{attribute 'GeneratedUsingTerminal: EJ7041-0052-0016'}
{attribute addProperty BoxType "EJ7041-0052-0016"}
{attribute addProperty Id "ENC_Status_compactAT %I*ENC_Status_compact_3C6E2C4411STM_StatusAT %I*STM_Status_36ED096F11ENC_Control_compactAT %Q*ENC_Control_compact_2E82BC435STM_ControlAT %Q*STM_Control_5A8B50163STM_VelocityAT %Q*STM_Velocity_A47A3F412WcStateAT %I*WcState_9091E0EB2InfoDataAT %I*InfoData_6538CF5F12"}
{attribute addProperty CRC "36390916"}
{attribute addProperty Size "46"}
TYPE EJ7041_022B4804 EXTENDS EtcSlaveTerminalBase_947E5A46 :
STRUCT
	{attribute addProperty Name "ENC_Status_compact"}
	ENC_Status_compact : ENC_Status_compact_3C6E2C44;
	{attribute addProperty Name "STM_Status"}
	STM_Status : STM_Status_36ED096F;
	{attribute addProperty Name "ENC_Control_compact"}
	ENC_Control_compact : ENC_Control_compact_2E82BC43;
	{attribute addProperty Name "STM_Control"}
	STM_Control : STM_Control_5A8B5016;
	{attribute addProperty Name "STM_Velocity"}
	STM_Velocity : STM_Velocity_A47A3F41;
	{attribute addProperty Name "WcState"}
	WcState : WcState_9091E0EB;
	{attribute addProperty Name "InfoData"}
	InfoData : InfoData_6538CF5F;
END_STRUCT
END_TYPE

(* stored: Version 1.2.0.0, ProductVersion 3.1.4024.9
   DUT EJ7041_022B4804: Id {041a55db-3422-4252-958e-5b21038afe5a} *)
